{attribute 'qualified_only'}
{attribute 'strict'}
{attribute 'To String'}
TYPE E_Devices :
(
	Undefined,
	Valve,
	Cylinder,
	Axis,
	PushButtonLight,
	DigitalSensor,
	AnalogSensor,
	DigitalOut,
	AnalogOut,
	PWMController,
	DoublePWMController,
	Encoder,
	AnalogAxis,
	TwoVelocityAxis,
	KL5151,
	KL1512
)INT;
END_TYPE

(* stored: Version 1.1.0.1, ProductVersion 3.1.4024.10
   EnumerationTextList E_Devices: Id {46bcbc51-0c54-0108-2c95-6d230f5291c3} *)
